// TIA Portal V18 export
TYPE "UDT_actualValues"
// stored: IsFailsafeCompliant false
   STRUCT
      target { ExternalVisible := 'False'; ExternalWritable := 'False'} : DInt;
      actual { ExternalVisible := 'False'; ExternalWritable := 'False'} : DInt;
      ok { ExternalVisible := 'False'; ExternalWritable := 'False'} : DInt;
      difference { ExternalVisible := 'False'; ExternalWritable := 'False'} : DInt;
      counterTactTime { ExternalVisible := 'False'; ExternalWritable := 'False'} : DInt;
      state { ExternalVisible := 'False'; ExternalWritable := 'False'} : DInt;
   END_STRUCT;
END_TYPE
